// TIA Portal V17 export
// export: Created 2024-09-03T21:54:56.631813Z, ExportSetting WithDefaults, DisplayName Totally Integrated Automation Portal, DisplayVersion V17 Update 7, DisplayName TIA Portal Openness, DisplayVersion V17 Update 7, DisplayName TIA Portal Version Control Interface, DisplayVersion V17, DisplayName SINAMICS Startdrive Advanced, DisplayVersion V17 SP2, DisplayName SINAMICS Startdrive G110M, G120, G120C, G120D, G120P, G115D, DisplayVersion V17 SP2, DisplayName SINAMICS Startdrive G130, G150, S120, S150, SINAMICS MV, S210, DisplayVersion V17 SP2, DisplayName STEP 7 Professional, DisplayVersion V17 Update 7, DisplayName STEP 7 Safety, DisplayVersion V17 Update 6, DisplayName WinCC Advanced / Unified PC, DisplayVersion V17 Update 7
DATA_BLOCK "AutoInfo"   // DB13
{ S7_Optimized_Access := 'TRUE' }
VERSION : 0.1
// stored: AutoNumber true, DBAccessibleFromOPCUA true, DBAccessibleFromWebserver true, IsOnlyStoredInLoadMemory false, IsRetainMemResEnabled false, IsWriteProtectedInAS false, MemoryReserve 100
   VAR
      EraseStation : Array[1..8] of Bool;
      ExtractedScan : String := '';
      EnableReferenceChange : Bool := TRUE;
   END_VAR
   VAR RETAIN
      R1BrakeTestRequired : Bool := TRUE;
      R1MasteringRequired : Bool := TRUE;
      PartMeasuredData { S7_SetPoint := 'True'} : "UDT_MeasuredPartData";
   END_VAR
   VAR
      EndProduction { S7_SetPoint := 'True'} : Bool;
   END_VAR
BEGIN
   EraseStation[1..8] := FALSE;
   PartMeasuredData.LeftCupforming.MaxForce := -7.98946;
   PartMeasuredData.LeftCupforming.MinimalWay := 9.841429;
   PartMeasuredData.LeftCupforming.MaxZposition := 55.44488;
   PartMeasuredData.LeftCupforming.OK := TRUE;
   PartMeasuredData.LeftCupforming.NOK := FALSE;
   PartMeasuredData.LeftCupforming.parameters.DigiforceProgram := 1;
   PartMeasuredData.LeftCupforming.parameters.FinalSpeed := 20.0;
   PartMeasuredData.LeftCupforming.parameters.ApproachSpeed := 100.0;
   PartMeasuredData.LeftCupforming.parameters.FinalForce := 80.0;
   PartMeasuredData.LeftCupforming.parameters.ApproachForce := 20.0;
   PartMeasuredData.LeftCupforming.parameters.EndWayImmediate := 9.9;
   PartMeasuredData.LeftCupforming.parameters.EndWayWithTimeout := 9.9;
   PartMeasuredData.LeftCupforming.parameters.SwitchingWay := 50.0;
   PartMeasuredData.LeftCupforming.parameters.EndWayTimeout := T#300MS;
   PartMeasuredData.RightCupforming.MaxForce := 8.163286;
   PartMeasuredData.RightCupforming.MinimalWay := 9.87697;
   PartMeasuredData.RightCupforming.MaxZposition := 56.52127;
   PartMeasuredData.RightCupforming.OK := TRUE;
   PartMeasuredData.RightCupforming.NOK := FALSE;
   PartMeasuredData.RightCupforming.parameters.DigiforceProgram := 1;
   PartMeasuredData.RightCupforming.parameters.FinalSpeed := 20.0;
   PartMeasuredData.RightCupforming.parameters.ApproachSpeed := 100.0;
   PartMeasuredData.RightCupforming.parameters.FinalForce := 80.0;
   PartMeasuredData.RightCupforming.parameters.ApproachForce := 20.0;
   PartMeasuredData.RightCupforming.parameters.EndWayImmediate := 9.9;
   PartMeasuredData.RightCupforming.parameters.EndWayWithTimeout := 9.9;
   PartMeasuredData.RightCupforming.parameters.SwitchingWay := 50.0;
   PartMeasuredData.RightCupforming.parameters.EndWayTimeout := T#300MS;
   PartMeasuredData.LeftRiveting1.Start := FALSE;
   PartMeasuredData.LeftRiveting1.PrgNumber := 0;
   PartMeasuredData.LeftRiveting1.Ready := FALSE;
   PartMeasuredData.LeftRiveting1.Running := FALSE;
   PartMeasuredData.LeftRiveting1.OK := FALSE;
   PartMeasuredData.LeftRiveting1.NOK := FALSE;
   PartMeasuredData.LeftRiveting1.H1OK := FALSE;
   PartMeasuredData.LeftRiveting1.H2OK := FALSE;
   PartMeasuredData.LeftRiveting1.TimeOK := FALSE;
   PartMeasuredData.LeftRiveting1.StartError := FALSE;
   PartMeasuredData.LeftRiveting1.LastH1 := 0.0;
   PartMeasuredData.LeftRiveting1.LastH2 := 0.0;
   PartMeasuredData.LeftRiveting1.LastTime := 0.0;
   PartMeasuredData.LeftRiveting1.LastZ1 := 0.0;
   PartMeasuredData.LeftRiveting1.Error := FALSE;
   PartMeasuredData.LeftRiveting1.NewData := FALSE;
   PartMeasuredData.LeftRiveting1.Z1OK := FALSE;
   PartMeasuredData.LeftRiveting1.NewDataAfterStart := FALSE;
   PartMeasuredData.LeftRiveting1.LastZ2 := 0.0;
   PartMeasuredData.LeftRiveting2.Start := FALSE;
   PartMeasuredData.LeftRiveting2.PrgNumber := 0;
   PartMeasuredData.LeftRiveting2.Ready := FALSE;
   PartMeasuredData.LeftRiveting2.Running := FALSE;
   PartMeasuredData.LeftRiveting2.OK := FALSE;
   PartMeasuredData.LeftRiveting2.NOK := FALSE;
   PartMeasuredData.LeftRiveting2.H1OK := FALSE;
   PartMeasuredData.LeftRiveting2.H2OK := FALSE;
   PartMeasuredData.LeftRiveting2.TimeOK := FALSE;
   PartMeasuredData.LeftRiveting2.StartError := FALSE;
   PartMeasuredData.LeftRiveting2.LastH1 := 0.0;
   PartMeasuredData.LeftRiveting2.LastH2 := 0.0;
   PartMeasuredData.LeftRiveting2.LastTime := 0.0;
   PartMeasuredData.LeftRiveting2.LastZ1 := 0.0;
   PartMeasuredData.LeftRiveting2.Error := FALSE;
   PartMeasuredData.LeftRiveting2.NewData := FALSE;
   PartMeasuredData.LeftRiveting2.Z1OK := FALSE;
   PartMeasuredData.LeftRiveting2.NewDataAfterStart := FALSE;
   PartMeasuredData.LeftRiveting2.LastZ2 := 0.0;
   PartMeasuredData.RightRiveting1.Start := FALSE;
   PartMeasuredData.RightRiveting1.PrgNumber := 0;
   PartMeasuredData.RightRiveting1.Ready := FALSE;
   PartMeasuredData.RightRiveting1.Running := FALSE;
   PartMeasuredData.RightRiveting1.OK := FALSE;
   PartMeasuredData.RightRiveting1.NOK := FALSE;
   PartMeasuredData.RightRiveting1.H1OK := FALSE;
   PartMeasuredData.RightRiveting1.H2OK := FALSE;
   PartMeasuredData.RightRiveting1.TimeOK := FALSE;
   PartMeasuredData.RightRiveting1.StartError := FALSE;
   PartMeasuredData.RightRiveting1.LastH1 := 0.0;
   PartMeasuredData.RightRiveting1.LastH2 := 0.0;
   PartMeasuredData.RightRiveting1.LastTime := 0.0;
   PartMeasuredData.RightRiveting1.LastZ1 := 0.0;
   PartMeasuredData.RightRiveting1.Error := FALSE;
   PartMeasuredData.RightRiveting1.NewData := FALSE;
   PartMeasuredData.RightRiveting1.Z1OK := FALSE;
   PartMeasuredData.RightRiveting1.NewDataAfterStart := FALSE;
   PartMeasuredData.RightRiveting1.LastZ2 := 0.0;
   PartMeasuredData.RightRiveting2.Start := FALSE;
   PartMeasuredData.RightRiveting2.PrgNumber := 0;
   PartMeasuredData.RightRiveting2.Ready := FALSE;
   PartMeasuredData.RightRiveting2.Running := FALSE;
   PartMeasuredData.RightRiveting2.OK := FALSE;
   PartMeasuredData.RightRiveting2.NOK := FALSE;
   PartMeasuredData.RightRiveting2.H1OK := FALSE;
   PartMeasuredData.RightRiveting2.H2OK := FALSE;
   PartMeasuredData.RightRiveting2.TimeOK := FALSE;
   PartMeasuredData.RightRiveting2.StartError := FALSE;
   PartMeasuredData.RightRiveting2.LastH1 := 0.0;
   PartMeasuredData.RightRiveting2.LastH2 := 0.0;
   PartMeasuredData.RightRiveting2.LastTime := 0.0;
   PartMeasuredData.RightRiveting2.LastZ1 := 0.0;
   PartMeasuredData.RightRiveting2.Error := FALSE;
   PartMeasuredData.RightRiveting2.NewData := FALSE;
   PartMeasuredData.RightRiveting2.Z1OK := FALSE;
   PartMeasuredData.RightRiveting2.NewDataAfterStart := FALSE;
   PartMeasuredData.RightRiveting2.LastZ2 := 0.0;
END_DATA_BLOCK
